PROGRAM MAIN
VAR
	fbFactorial : IO.Factorial;
	fbFactorial_2 : IO.Factorial;
END_VAR

fbFactorial(); 
fbFactorial_2();

END_PROGRAM

(* stored: Version 1.1.0.1, ProductVersion 3.1.4024.12
   POU MAIN: Id {e02ffb5a-bf0c-4392-8a13-b0306996ad4d}, SpecialFunc None *)
